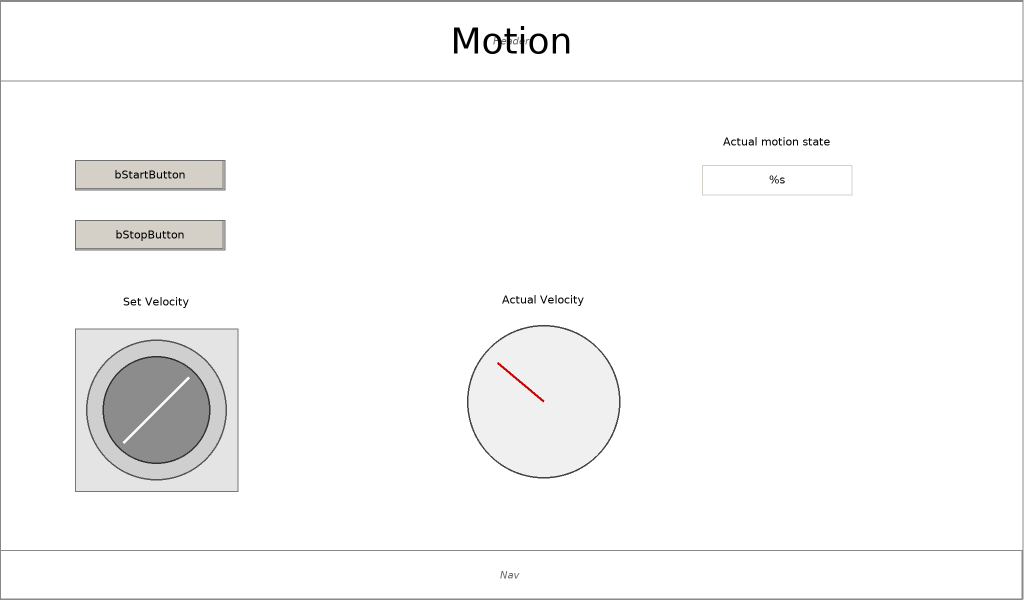
VISUALIZATION Motion  // 1024x600
    Frame (-1,1 1024x80)
        shows Header()
    Frame (-2,550 1024x50)
        shows Nav()
    Label (333,17 357x48), "Motion"
    Textfield (702,165 150x30), "%s", text variable: Motion.sMotionState
    Label (702,127 150x30), "Actual motion state"
    Button (75,160 150x30), "bStartButton"
        OnMouseDown: execute { Motion.bStartButton := TRUE; }
        OnMouseUp: execute { Motion.bStartButton := FALSE; }
    Button (75,220 150x30), "bStopButton"
        OnMouseDown: execute { Motion.bStopButton := TRUE; }
        OnMouseUp: execute { Motion.bStopButton := FALSE; }
    Potentiometer360 (75,325 163x170), variable: Motion.SetVelocity, style: Potentiometer-Potentiometer360-Gray, scale format: %.1f, scale 0..4000
        p2431819421: Outside
    Meter360 (465,325 157x153), value: Motion.Axis1.NcToPlc.ActVelo, style: Meter-Meter360-Gray, scale format: %5.2f, scale 0..4000
    Label (81,287 150x30), "Set Velocity"
    Label (468,285 150x30), "Actual Velocity"
END_VISUALIZATION

(* stored: Version 1.1.0.1, ProductVersion 3.1.4024.12
   Visu Motion: Id {c5b5a224-37b0-4f7a-a46c-71d675aef9cb} *)
